{attribute 'GeneratedUsingTerminal: EL2212-0000-0020'}
{attribute addProperty BoxType "EL2212-0000-0020"}
{attribute addProperty Id "DOX_Status_Channel_1AT %I*DOX_Status_Channel_6FDDBA987DOX_Status_Channel_2AT %I*DOX_Status_Channel_6FDDBA987DOX_Control_Channel_1AT %Q*DOX_Control_Channel_E69306414DOX_Control_Channel_2AT %Q*DOX_Control_Channel_E69306414WcStateAT %I*WcState_9091E0EB2InfoDataAT %I*InfoData_94A18F5E2"}
{attribute addProperty CRC "274588809"}
{attribute addProperty Size "26"}
TYPE EL2212_105DE489 EXTENDS EtcSlaveTerminalBase_947E5A46 :
STRUCT
	{attribute addProperty Name "DOX_Status_Channel_1"}
	DOX_Status_Channel_1 : DOX_Status_Channel_6FDDBA98;
	{attribute addProperty Name "DOX_Status_Channel_2"}
	DOX_Status_Channel_2 : DOX_Status_Channel_6FDDBA98;
	{attribute addProperty Name "DOX_Control_Channel_1"}
	DOX_Control_Channel_1 : DOX_Control_Channel_E6930641;
	{attribute addProperty Name "DOX_Control_Channel_2"}
	DOX_Control_Channel_2 : DOX_Control_Channel_E6930641;
	{attribute addProperty Name "WcState"}
	WcState : WcState_9091E0EB;
	{attribute addProperty Name "InfoData"}
	InfoData : InfoData_94A18F5E;
END_STRUCT
END_TYPE

(* stored: Version 1.2.0.0, ProductVersion 3.1.4024.9
   DUT EL2212_105DE489: Id {ebd6ac7a-a07a-4f26-936b-007b9449977a} *)
